Staubli VAL3: PentagonPoint.pgx

public program PentagonPoint(trsf& x_trSource[], trsf& x_trDest[], bool& x_bRes)
  local point l_pPoint[3]
  local num l_ni
  local frame l_fFrame
  local num l_Dia
  local num l_nLegth
  local point l_pBuff
begin
  //五边形
  //根据三个trsf建立frame
  call SetFrame(x_trSource,l_fFrame,x_bRes)
  if !x_bRes
    return
  endIf

  //圆弧的直径
//  l_Dia=distance(x_trSource[1],x_trSource[2])
  l_nLegth=distance(x_trSource[0],x_trSource[1])



  link(l_pBuff,l_fFrame)
  l_pBuff.trsf={l_nLegth/2,0,0,0,0,0}
  x_trDest[0]=position(l_pBuff,world)

  l_pBuff.trsf={l_nLegth,0,0,0,0,0}
  x_trDest[1]=position(l_pBuff,world)

//  l_pBuff.trsf={l_nLegth+sin(18)*l_nLegth,cos(18)*l_nLegth,0,0,0,0}
//  x_trDest[2]=position(l_pBuff,world)
//
//  l_pBuff.trsf={l_nLegth/2,(sin(36)+sin(54))*l_nLegth,0,0,0,0}
//  x_trDest[3]=position(l_pBuff,world)
//
//  l_pBuff.trsf={-sin(36)*l_nLegth,cos(36)*l_nLegth,0,0,0,0}
//  x_trDest[4]=position(l_pBuff,world)
//

//2013.10.26
  l_pBuff.trsf={l_nLegth+sin(18)*l_nLegth,cos(18)*l_nLegth,0,0,0,0}
  x_trDest[2]=position(l_pBuff,world)

  l_pBuff.trsf={l_nLegth/2,(sin(36)+sin(72))*l_nLegth,0,0,0,0}
  x_trDest[3]=position(l_pBuff,world)

  l_pBuff.trsf={-sin(18)*l_nLegth,cos(18)*l_nLegth,0,0,0,0}
  x_trDest[4]=position(l_pBuff,world)




//*************************************

  l_pBuff.trsf={0,0,0,0,0,0}
  x_trDest[5]=position(l_pBuff,world)

  x_trDest[6]=x_trDest[0]

    //圆心点
  l_pBuff.trsf={l_nLegth/2,l_nLegth/2/sin(36),0,0,0,0}
  x_trDest[20]=position(l_pBuff,world)



end
